PROGRAM SDODaten
VAR
	DatenMotor1: SDODatenMotor1;
	DatenMotor2: SDODatenMotor2;
	DatenMotor3: SDODatenMotor3;
	DatenMotorklemme1: SDODatenMotorklemme1;
	DatenMotorklemme2: SDODatenMotorklemme2;
END_VAR

DatenMotor1();
DatenMotor2();
DatenMotor3();
DatenMotorklemme1();
DatenMotorklemme2();

END_PROGRAM

(* stored: Version 1.1.0.1, ProductVersion 3.1.4020.12
   POU SDODaten: Id {4be8eb0e-eb8a-4a8c-aa30-ca78f43e7d4b}, SpecialFunc None *)
